(* CoDeSys 2.3 export: ERRORENTRY_TS.EXP *)

(* Data type in Diag/Error *)
TYPE ErrorEntry_ts :
STRUCT
	Code_u16					: UINT;
	Param_u8					: USINT;
	Frequency_u8			: USINT;
	TimeStamp_u32			: UDINT;
END_STRUCT
END_TYPE
